PROGRAM MAIN
VAR
END_VAR

END_PROGRAM

(* stored: Version 1.1.0.1
   POU MAIN: Id {012c14aa-93d3-4c2d-99f0-18f228a90f72} *)
